# EPICS autosave request: iocBoot/ioc6bmb/Galil_positions.req
file "CARS_24_motor_positions.req",    P=$(P)
